TYPE csp_transfer_upstacker_test_status_enum :
(		
	CSP_TRANSFER_UPSTACKER_STATUS_TEST_START								:= 0,
	CSP_TRANSFER_UPSTACKER_STATUS_TEST_DISABLE 								:= 10,
	CSP_TRANSFER_UPSTACKER_STATUS_TEST_ENABLE 								:= 20,
	CSP_TRANSFER_UPSTACKER_STATUS_TEST_ENABLED								:= 30,
	CSP_TRANSFER_UPSTACKER_STATUS_TEST_JOG_DOWNSTREAM						:= 40,
	CSP_TRANSFER_UPSTACKER_STATUS_TEST_REDEFINE_DOWNSTREAM					:= 50,
	CSP_TRANSFER_UPSTACKER_STATUS_TEST_JOG_UPSTREAM							:= 60,
	CSP_TRANSFER_UPSTACKER_STATUS_TEST_REDEFINE_UPSTREAM					:= 70,
	CSP_TRANSFER_UPSTACKER_STATUS_TEST_STOP 								:= 80,
	CSP_TRANSFER_UPSTACKER_STATUS_TEST_ERROR 								:= 999
) := CSP_TRANSFER_UPSTACKER_STATUS_TEST_START;
END_TYPE

(* stored: Version 1.1.0.1, ProductVersion 3.1.4022.12
   DUT csp_transfer_upstacker_test_status_enum: Id {24db007f-f4ef-4f6c-8fe1-41528ab8a54b} *)
